KUKA KRL program: ps_b_ltb_res_c03.src, ps_b_ltb_res_c03.dat

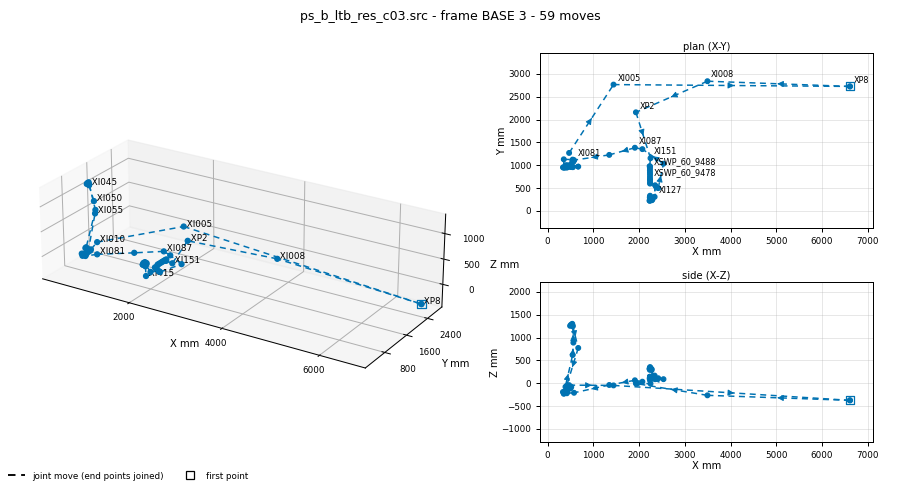
[picture p0: tool path of ps_b_ltb_res_c03.src in frame BASE 3, 59 of 59 moves have a stored position in this frame; points joined in program order, loops and branches not executed]
--- ps_b_ltb_res_c03.src ---
&ACCESS RVO1
&COMMENT Solda Atego LTB
&PARAM DISKPATH = KRC:\R1\Program\inpro_nao_mexer
DEF ps_b_ltb_res_c03( )
;FOLD INI
;FOLD SPOTTECH INI
USERSPOT(#INIT)
;ENDFOLD (SPOTTECH INI)
;FOLD GRIPPERTECH INI
USER_GRP(0,DUMMY,DUMMY,GDEFAULT)
;ENDFOLD (GRIPPERTECH INI)
  ;FOLD USER INI
    ;Make your modifications here

  ;ENDFOLD (USER INI)
;ENDFOLD (INI)

; Caracterizacao dos meios de producao
; Changes: Solda Respot - ATEGO LTB
; Versao Atual:29/10/2016
; Ferramenta: Gun C3
; Name: P13.050-R2
; optimisation

chk_w4_wechs_ok( )      ; CHECK GUN C3

;FOLD PTP P8 Vel=100 % PDAT4 Tool[4]:Gun C3 Base[3]:Atego/Axor;%{PE}%R 8.2.20,%MKUKATPBASIS,%CMOVE,%VPTP,%P 1:PTP, 2:P8, 3:, 5:100, 7:PDAT4
$BWDSTART=FALSE
PDAT_ACT=PPDAT4
FDAT_ACT=FP8
BAS(#PTP_PARAMS,100)
PTP XP8
;ENDFOLD

if MaxStandMenge (3) then
 MaxStandmengeErreicht (3)
endif

 IF (NOT(GHOST())) THEN
 if FraesAnf (3) then
 e_fraes4 ()
 endif
 ENDIF

;FOLD PTP l008 Vel=100 % P_OLP13 Tool[4]:Gun C3 Base[3]:Atego/Axor;%{PE}%R 8.2.20,%MKUKATPBASIS,%CMOVE,%VPTP,%P 1:PTP, 2:l008, 3:, 5:100, 7:P_OLP13
$BWDSTART=FALSE
PDAT_ACT=PP_OLP13
FDAT_ACT=Fl008
BAS(#PTP_PARAMS,100)
PTP Xl008
;ENDFOLD

; AGUARDA LIBERACAO PARA SOLDAR RESPOT
;FOLD OUT 3338 'R2 solda geometria Ok' State=FALSE ;%{PE}%R 8.2.20,%MKUKATPBASIS,%COUT,%VOUTX,%P 2:3338, 3:R2 solda geometria Ok, 5:FALSE, 6:
$OUT[3338]=FALSE
;ENDFOLD
;FOLD OUT 3348 'Fora area GEOBOX' State=FALSE ;%{PE}%R 8.2.20,%MKUKATPBASIS,%COUT,%VOUTX,%P 2:3348, 3:Fora area GEOBOX, 5:FALSE, 6:
$OUT[3348]=FALSE
;ENDFOLD
;FOLD OUT 3380 'Lib. p/ soldar Res Axor/Atego' State=TRUE ;%{PE}%R 8.2.20,%MKUKATPBASIS,%COUT,%VOUTX,%P 2:3380, 3:Lib. p/ soldar Res Axor/Atego, 5:TRUE, 6:
$OUT[3380]=TRUE
;ENDFOLD
;FOLD WAIT FOR ( IN 3380 'Lib. p/ soldar Res Axor/Atego' );%{PE}%R 8.2.20,%MKUKATPBASIS,%CEXT_WAIT_FOR,%VEXT_WAIT_FOR,%P 2:, 4:, 5:$IN, 6:3380, 7:Lib. p/ soldar Res Axor/Atego, 9:
WAIT FOR  ( $IN[3380] )
;ENDFOLD
;FOLD OUT 3380 'Lib. p/ soldar Res Axor/Atego' State=FALSE ;%{PE}%R 8.2.20,%MKUKATPBASIS,%COUT,%VOUTX,%P 2:3380, 3:Lib. p/ soldar Res Axor/Atego, 5:FALSE, 6:
$OUT[3380]=FALSE
;ENDFOLD

; LIGA INTERTRAVAMENTO 1 C/ R1
;FOLD Collision.Monitoring_1_On ;%{PE}%MKUKATPUSER
COLLSTOP( 1, 1 ) ;Interrupt-Controlled
;ENDFOLD

; LIGA INTERTRAVAMENTO 4 C/ R4
;FOLD Collision.Monitoring_4_On ;%{PE}%MKUKATPUSER
COLLSTOP( 4, 1 ) ;Interrupt-Controlled
;ENDFOLD

;FOLD PTP P2 CONT Vel=100 % xlarge Tool[4]:Gun C3 Base[3]:Atego/Axor;%{PE}%R 8.2.20,%MKUKATPBASIS,%CMOVE,%VPTP,%P 1:PTP, 2:P2, 3:C_DIS, 5:100, 7:xlarge
$BWDSTART=FALSE
PDAT_ACT=Pxlarge
FDAT_ACT=FP2
BAS(#PTP_PARAMS,100)
PTP XP2 C_DIS
;ENDFOLD
;FOLD PTP l151 CONT Vel=100 % large Tool[4]:Gun C3 Base[3]:Atego/Axor;%{PE}%R 8.2.20,%MKUKATPBASIS,%CMOVE,%VPTP,%P 1:PTP, 2:l151, 3:C_DIS, 5:100, 7:large
$BWDSTART=FALSE
PDAT_ACT=Plarge
FDAT_ACT=Fl151
BAS(#PTP_PARAMS,100)
PTP Xl151 C_DIS
;ENDFOLD
;FOLD PTP l146 CONT Vel=100 % fin Tool[4]:Gun C3 Base[3]:Atego/Axor;%{PE}%R 8.2.20,%MKUKATPBASIS,%CMOVE,%VPTP,%P 1:PTP, 2:l146, 3:C_DIS, 5:100, 7:fin
$BWDSTART=FALSE
PDAT_ACT=Pfin
FDAT_ACT=Fl146
BAS(#PTP_PARAMS,100)
PTP Xl146 C_DIS
;ENDFOLD

;FOLD ; SWP_60_9490;%{PE}%R 8.2.20,%MKUKATPBASIS,%CCOMMENT,%VNORMAL,%P 2:SWP_60_9490
;ENDFOLD
;FOLD PTP SWP_60_9490 vmax SPOT Gun=3 RETR CLS PgNo1=199 ACTIVE=1 Tool[4]:Gun C3 Base[3]:Atego/Axor;%{PE}%R 8.2.2,%MKUKATPSPOT,%CSPOT,%VPTP,%P 1:PTP, 2:SWP_60_9490, 3:, 5:100, 7:vmax, 10:3, 12:#FIRST, 14:#CLO, 16:199, 18:1, 20:0, 22:0, 24:1, 25:NORMAL
$BWDSTART=FALSE
PDAT_ACT=Pvmax
FDAT_ACT=FSWP_60_9490
BAS(#PTP_PARAMS,Pvmax.VEL)
S_ACT.GUN=3
S_ACT.PAIR=SDEFAULT.PAIR
S_ACT.RETR=#CLO
S_ACT.CLO_TM=1
S_ACT.PGNO1=199
S_ACT.PGNO2=SDEFAULT.PGNO2
S_ACT.PRESS1=SDEFAULT.PRESS1
S_ACT.PRESS2=SDEFAULT.PRESS2
S_READY=FALSE
PTP XSWP_60_9490
USERSPOT(#SPOT, S_ACT)
WAIT FOR S_READY
;ENDFOLD

;FOLD ; SWP_60_9488;%{PE}%R 8.2.20,%MKUKATPBASIS,%CCOMMENT,%VNORMAL,%P 2:SWP_60_9488
;ENDFOLD
;FOLD PTP SWP_60_9488 vmax SPOT Gun=3 RETR CLS PgNo1=199 ACTIVE=1 Tool[4]:Gun C3 Base[3]:Atego/Axor;%{PE}%R 8.2.2,%MKUKATPSPOT,%CSPOT,%VPTP,%P 1:PTP, 2:SWP_60_9488, 3:, 5:100, 7:vmax, 10:3, 12:#FIRST, 14:#CLO, 16:199, 18:1, 20:0, 22:0, 24:1, 25:NORMAL
$BWDSTART=FALSE
PDAT_ACT=Pvmax
FDAT_ACT=FSWP_60_9488
BAS(#PTP_PARAMS,Pvmax.VEL)
S_ACT.GUN=3
S_ACT.PAIR=SDEFAULT.PAIR
S_ACT.RETR=#CLO
S_ACT.CLO_TM=1
S_ACT.PGNO1=199
S_ACT.PGNO2=SDEFAULT.PGNO2
S_ACT.PRESS1=SDEFAULT.PRESS1
S_ACT.PRESS2=SDEFAULT.PRESS2
S_READY=FALSE
PTP XSWP_60_9488
USERSPOT(#SPOT, S_ACT)
WAIT FOR S_READY
;ENDFOLD

;FOLD ; SWP_60_9486;%{PE}%R 8.2.20,%MKUKATPBASIS,%CCOMMENT,%VNORMAL,%P 2:SWP_60_9486
;ENDFOLD
;FOLD PTP SWP_60_9486 vmax SPOT Gun=3 RETR CLS PgNo1=199 ACTIVE=1 Tool[4]:Gun C3 Base[3]:Atego/Axor;%{PE}%R 8.2.2,%MKUKATPSPOT,%CSPOT,%VPTP,%P 1:PTP, 2:SWP_60_9486, 3:, 5:100, 7:vmax, 10:3, 12:#FIRST, 14:#CLO, 16:199, 18:1, 20:0, 22:0, 24:1, 25:NORMAL
$BWDSTART=FALSE
PDAT_ACT=Pvmax
FDAT_ACT=FSWP_60_9486
BAS(#PTP_PARAMS,Pvmax.VEL)
S_ACT.GUN=3
S_ACT.PAIR=SDEFAULT.PAIR
S_ACT.RETR=#CLO
S_ACT.CLO_TM=1
S_ACT.PGNO1=199
S_ACT.PGNO2=SDEFAULT.PGNO2
S_ACT.PRESS1=SDEFAULT.PRESS1
S_ACT.PRESS2=SDEFAULT.PRESS2
S_READY=FALSE
PTP XSWP_60_9486
USERSPOT(#SPOT, S_ACT)
WAIT FOR S_READY
;ENDFOLD

;FOLD ; SWP_60_9484;%{PE}%R 8.2.20,%MKUKATPBASIS,%CCOMMENT,%VNORMAL,%P 2:SWP_60_9484
;ENDFOLD
;FOLD PTP SWP_60_9484 vmax SPOT Gun=3 RETR CLS PgNo1=199 ACTIVE=1 Tool[4]:Gun C3 Base[3]:Atego/Axor;%{PE}%R 8.2.2,%MKUKATPSPOT,%CSPOT,%VPTP,%P 1:PTP, 2:SWP_60_9484, 3:, 5:100, 7:vmax, 10:3, 12:#FIRST, 14:#CLO, 16:199, 18:1, 20:0, 22:0, 24:1, 25:NORMAL
$BWDSTART=FALSE
PDAT_ACT=Pvmax
FDAT_ACT=FSWP_60_9484
BAS(#PTP_PARAMS,Pvmax.VEL)
S_ACT.GUN=3
S_ACT.PAIR=SDEFAULT.PAIR
S_ACT.RETR=#CLO
S_ACT.CLO_TM=1
S_ACT.PGNO1=199
S_ACT.PGNO2=SDEFAULT.PGNO2
S_ACT.PRESS1=SDEFAULT.PRESS1
S_ACT.PRESS2=SDEFAULT.PRESS2
S_READY=FALSE
PTP XSWP_60_9484
USERSPOT(#SPOT, S_ACT)
WAIT FOR S_READY
;ENDFOLD

;FOLD ; SWP_60_9482;%{PE}%R 8.2.20,%MKUKATPBASIS,%CCOMMENT,%VNORMAL,%P 2:SWP_60_9482
;ENDFOLD
;FOLD PTP SWP_60_9482 vmax SPOT Gun=3 RETR CLS PgNo1=199 ACTIVE=1 Tool[4]:Gun C3 Base[3]:Atego/Axor;%{PE}%R 8.2.2,%MKUKATPSPOT,%CSPOT,%VPTP,%P 1:PTP, 2:SWP_60_9482, 3:, 5:100, 7:vmax, 10:3, 12:#FIRST, 14:#CLO, 16:199, 18:1, 20:0, 22:0, 24:1, 25:NORMAL
$BWDSTART=FALSE
PDAT_ACT=Pvmax
FDAT_ACT=FSWP_60_9482
BAS(#PTP_PARAMS,Pvmax.VEL)
S_ACT.GUN=3
S_ACT.PAIR=SDEFAULT.PAIR
S_ACT.RETR=#CLO
S_ACT.CLO_TM=1
S_ACT.PGNO1=199
S_ACT.PGNO2=SDEFAULT.PGNO2
S_ACT.PRESS1=SDEFAULT.PRESS1
S_ACT.PRESS2=SDEFAULT.PRESS2
S_READY=FALSE
PTP XSWP_60_9482
USERSPOT(#SPOT, S_ACT)
WAIT FOR S_READY
;ENDFOLD

;FOLD ; SWP_60_9480;%{PE}%R 8.2.20,%MKUKATPBASIS,%CCOMMENT,%VNORMAL,%P 2:SWP_60_9480
;ENDFOLD
;FOLD PTP SWP_60_9480 vmax SPOT Gun=3 RETR CLS PgNo1=199 ACTIVE=1 Tool[4]:Gun C3 Base[3]:Atego/Axor;%{PE}%R 8.2.2,%MKUKATPSPOT,%CSPOT,%VPTP,%P 1:PTP, 2:SWP_60_9480, 3:, 5:100, 7:vmax, 10:3, 12:#FIRST, 14:#CLO, 16:199, 18:1, 20:0, 22:0, 24:1, 25:NORMAL
$BWDSTART=FALSE
PDAT_ACT=Pvmax
FDAT_ACT=FSWP_60_9480
BAS(#PTP_PARAMS,Pvmax.VEL)
S_ACT.GUN=3
S_ACT.PAIR=SDEFAULT.PAIR
S_ACT.RETR=#CLO
S_ACT.CLO_TM=1
S_ACT.PGNO1=199
S_ACT.PGNO2=SDEFAULT.PGNO2
S_ACT.PRESS1=SDEFAULT.PRESS1
S_ACT.PRESS2=SDEFAULT.PRESS2
S_READY=FALSE
PTP XSWP_60_9480
USERSPOT(#SPOT, S_ACT)
WAIT FOR S_READY
;ENDFOLD

;FOLD ; SWP_60_9478;%{PE}%R 8.2.20,%MKUKATPBASIS,%CCOMMENT,%VNORMAL,%P 2:SWP_60_9478
;ENDFOLD
;FOLD PTP SWP_60_9478 vmax SPOT Gun=3 RETR CLS PgNo1=199 ACTIVE=1 Tool[4]:Gun C3 Base[3]:Atego/Axor;%{PE}%R 8.2.2,%MKUKATPSPOT,%CSPOT,%VPTP,%P 1:PTP, 2:SWP_60_9478, 3:, 5:100, 7:vmax, 10:3, 12:#FIRST, 14:#CLO, 16:199, 18:1, 20:0, 22:0, 24:1, 25:NORMAL
$BWDSTART=FALSE
PDAT_ACT=Pvmax
FDAT_ACT=FSWP_60_9478
BAS(#PTP_PARAMS,Pvmax.VEL)
S_ACT.GUN=3
S_ACT.PAIR=SDEFAULT.PAIR
S_ACT.RETR=#CLO
S_ACT.CLO_TM=1
S_ACT.PGNO1=199
S_ACT.PGNO2=SDEFAULT.PGNO2
S_ACT.PRESS1=SDEFAULT.PRESS1
S_ACT.PRESS2=SDEFAULT.PRESS2
S_READY=FALSE
PTP XSWP_60_9478
USERSPOT(#SPOT, S_ACT)
WAIT FOR S_READY
;ENDFOLD

;FOLD PTP l140 CONT Vel=100 % fin Tool[4]:Gun C3 Base[3]:Atego/Axor;%{PE}%R 8.2.20,%MKUKATPBASIS,%CMOVE,%VPTP,%P 1:PTP, 2:l140, 3:C_DIS, 5:100, 7:fin
$BWDSTART=FALSE
PDAT_ACT=Pfin
FDAT_ACT=Fl140
BAS(#PTP_PARAMS,100)
PTP Xl140 C_DIS
;ENDFOLD

;FOLD ; SWP_60_9474;%{PE}%R 8.2.20,%MKUKATPBASIS,%CCOMMENT,%VNORMAL,%P 2:SWP_60_9474
;ENDFOLD
;FOLD PTP SWP_60_9474 vmax SPOT Gun=3 RETR CLS PgNo1=199 ACTIVE=1 Tool[4]:Gun C3 Base[3]:Atego/Axor;%{PE}%R 8.2.2,%MKUKATPSPOT,%CSPOT,%VPTP,%P 1:PTP, 2:SWP_60_9474, 3:, 5:100, 7:vmax, 10:3, 12:#FIRST, 14:#CLO, 16:199, 18:1, 20:0, 22:0, 24:1, 25:NORMAL
$BWDSTART=FALSE
PDAT_ACT=Pvmax
FDAT_ACT=FSWP_60_9474
BAS(#PTP_PARAMS,Pvmax.VEL)
S_ACT.GUN=3
S_ACT.PAIR=SDEFAULT.PAIR
S_ACT.RETR=#CLO
S_ACT.CLO_TM=1
S_ACT.PGNO1=199
S_ACT.PGNO2=SDEFAULT.PGNO2
S_ACT.PRESS1=SDEFAULT.PRESS1
S_ACT.PRESS2=SDEFAULT.PRESS2
S_READY=FALSE
PTP XSWP_60_9474
USERSPOT(#SPOT, S_ACT)
WAIT FOR S_READY
;ENDFOLD

; LIGA INTERTRAVAMENTO 12 C/ R1
;FOLD Collision.Monitoring_AREA_6_On ;%{PE}%MKUKATPUSER
COLLSTOP( 12, 1 ) ;not Interrupt-Controlled
;ENDFOLD

;FOLD PTP l131 CONT Vel=100 % fin Tool[4]:Gun C3 Base[3]:Atego/Axor;%{PE}%R 8.2.20,%MKUKATPBASIS,%CMOVE,%VPTP,%P 1:PTP, 2:l131, 3:C_DIS, 5:100, 7:fin
$BWDSTART=FALSE
PDAT_ACT=Pfin
FDAT_ACT=Fl131
BAS(#PTP_PARAMS,100)
PTP Xl131 C_DIS
;ENDFOLD
;FOLD PTP l126 CONT Vel=100 % small Tool[4]:Gun C3 Base[3]:Atego/Axor;%{PE}%R 8.2.20,%MKUKATPBASIS,%CMOVE,%VPTP,%P 1:PTP, 2:l126, 3:C_DIS, 5:100, 7:small
$BWDSTART=FALSE
PDAT_ACT=Psmall
FDAT_ACT=Fl126
BAS(#PTP_PARAMS,100)
PTP Xl126 C_DIS
;ENDFOLD
;FOLD PTP l127 CONT Vel=100 % small Tool[4]:Gun C3 Base[3]:Atego/Axor;%{PE}%R 8.2.20,%MKUKATPBASIS,%CMOVE,%VPTP,%P 1:PTP, 2:l127, 3:C_DIS, 5:100, 7:small
$BWDSTART=FALSE
PDAT_ACT=Psmall
FDAT_ACT=Fl127
BAS(#PTP_PARAMS,100)
PTP Xl127 C_DIS
;ENDFOLD
;FOLD PTP l128 CONT Vel=100 % fin Tool[4]:Gun C3 Base[3]:Atego/Axor;%{PE}%R 8.2.20,%MKUKATPBASIS,%CMOVE,%VPTP,%P 1:PTP, 2:l128, 3:C_DIS, 5:100, 7:fin
$BWDSTART=FALSE
PDAT_ACT=Pfin
FDAT_ACT=Fl128
BAS(#PTP_PARAMS,100)
PTP Xl128 C_DIS
;ENDFOLD

;FOLD ; SWP_60_9470;%{PE}%R 8.2.20,%MKUKATPBASIS,%CCOMMENT,%VNORMAL,%P 2:SWP_60_9470
;ENDFOLD
;FOLD PTP SWP_60_9470 vmax SPOT Gun=3 RETR CLS PgNo1=199 ACTIVE=1 Tool[4]:Gun C3 Base[3]:Atego/Axor;%{PE}%R 8.2.2,%MKUKATPSPOT,%CSPOT,%VPTP,%P 1:PTP, 2:SWP_60_9470, 3:, 5:100, 7:vmax, 10:3, 12:#FIRST, 14:#CLO, 16:199, 18:1, 20:0, 22:0, 24:1, 25:NORMAL
$BWDSTART=FALSE
PDAT_ACT=Pvmax
FDAT_ACT=FSWP_60_9470
BAS(#PTP_PARAMS,Pvmax.VEL)
S_ACT.GUN=3
S_ACT.PAIR=SDEFAULT.PAIR
S_ACT.RETR=#CLO
S_ACT.CLO_TM=1
S_ACT.PGNO1=199
S_ACT.PGNO2=SDEFAULT.PGNO2
S_ACT.PRESS1=SDEFAULT.PRESS1
S_ACT.PRESS2=SDEFAULT.PRESS2
S_READY=FALSE
PTP XSWP_60_9470
USERSPOT(#SPOT, S_ACT)
WAIT FOR S_READY
;ENDFOLD

;FOLD ; SWP_60_9468;%{PE}%R 8.2.20,%MKUKATPBASIS,%CCOMMENT,%VNORMAL,%P 2:SWP_60_9468
;ENDFOLD
;FOLD PTP SWP_60_9468 vmax SPOT Gun=3 RETR CLS PgNo1=199 ACTIVE=1 Tool[4]:Gun C3 Base[3]:Atego/Axor;%{PE}%R 8.2.2,%MKUKATPSPOT,%CSPOT,%VPTP,%P 1:PTP, 2:SWP_60_9468, 3:, 5:100, 7:vmax, 10:3, 12:#FIRST, 14:#CLO, 16:199, 18:1, 20:0, 22:0, 24:1, 25:NORMAL
$BWDSTART=FALSE
PDAT_ACT=Pvmax
FDAT_ACT=FSWP_60_9468
BAS(#PTP_PARAMS,Pvmax.VEL)
S_ACT.GUN=3
S_ACT.PAIR=SDEFAULT.PAIR
S_ACT.RETR=#CLO
S_ACT.CLO_TM=1
S_ACT.PGNO1=199
S_ACT.PGNO2=SDEFAULT.PGNO2
S_ACT.PRESS1=SDEFAULT.PRESS1
S_ACT.PRESS2=SDEFAULT.PRESS2
S_READY=FALSE
PTP XSWP_60_9468
USERSPOT(#SPOT, S_ACT)
WAIT FOR S_READY
;ENDFOLD

;FOLD PTP l129 CONT Vel=100 % fin Tool[4]:Gun C3 Base[3]:Atego/Axor;%{PE}%R 8.2.20,%MKUKATPBASIS,%CMOVE,%VPTP,%P 1:PTP, 2:l129, 3:C_DIS, 5:100, 7:fin
$BWDSTART=FALSE
PDAT_ACT=Pfin
FDAT_ACT=Fl129
BAS(#PTP_PARAMS,100)
PTP Xl129 C_DIS
;ENDFOLD
;FOLD PTP l130 CONT Vel=100 % fin Tool[4]:Gun C3 Base[3]:Atego/Axor;%{PE}%R 8.2.20,%MKUKATPBASIS,%CMOVE,%VPTP,%P 1:PTP, 2:l130, 3:C_DIS, 5:100, 7:fin
$BWDSTART=FALSE
PDAT_ACT=Pfin
FDAT_ACT=Fl130
BAS(#PTP_PARAMS,100)
PTP Xl130 C_DIS
;ENDFOLD
;FOLD PTP l132 CONT Vel=100 % fin Tool[4]:Gun C3 Base[3]:Atego/Axor;%{PE}%R 8.2.20,%MKUKATPBASIS,%CMOVE,%VPTP,%P 1:PTP, 2:l132, 3:C_DIS, 5:100, 7:fin
$BWDSTART=FALSE
PDAT_ACT=Pfin
FDAT_ACT=Fl132
BAS(#PTP_PARAMS,100)
PTP Xl132 C_DIS
;ENDFOLD
;FOLD PTP l133 CONT Vel=100 % fin Tool[4]:Gun C3 Base[3]:Atego/Axor;%{PE}%R 8.2.20,%MKUKATPBASIS,%CMOVE,%VPTP,%P 1:PTP, 2:l133, 3:C_DIS, 5:100, 7:fin
$BWDSTART=FALSE
PDAT_ACT=Pfin
FDAT_ACT=Fl133
BAS(#PTP_PARAMS,100)
PTP Xl133 C_DIS
;ENDFOLD

;FOLD ; SWP_60_9466;%{PE}%R 8.2.20,%MKUKATPBASIS,%CCOMMENT,%VNORMAL,%P 2:SWP_60_9466
;ENDFOLD
;FOLD PTP SWP_60_9466 vmax SPOT Gun=3 RETR CLS PgNo1=199 ACTIVE=1 Tool[4]:Gun C3 Base[3]:Atego/Axor;%{PE}%R 8.2.2,%MKUKATPSPOT,%CSPOT,%VPTP,%P 1:PTP, 2:SWP_60_9466, 3:, 5:100, 7:vmax, 10:3, 12:#FIRST, 14:#CLO, 16:199, 18:1, 20:0, 22:0, 24:1, 25:NORMAL
$BWDSTART=FALSE
PDAT_ACT=Pvmax
FDAT_ACT=FSWP_60_9466
BAS(#PTP_PARAMS,Pvmax.VEL)
S_ACT.GUN=3
S_ACT.PAIR=SDEFAULT.PAIR
S_ACT.RETR=#CLO
S_ACT.CLO_TM=1
S_ACT.PGNO1=199
S_ACT.PGNO2=SDEFAULT.PGNO2
S_ACT.PRESS1=SDEFAULT.PRESS1
S_ACT.PRESS2=SDEFAULT.PRESS2
S_READY=FALSE
PTP XSWP_60_9466
USERSPOT(#SPOT, S_ACT)
WAIT FOR S_READY
;ENDFOLD


;FOLD PTP l134 CONT Vel=100 % fin Tool[4]:Gun C3 Base[3]:Atego/Axor;%{PE}%R 8.2.20,%MKUKATPBASIS,%CMOVE,%VPTP,%P 1:PTP, 2:l134, 3:C_DIS, 5:100, 7:fin
$BWDSTART=FALSE
PDAT_ACT=Pfin
FDAT_ACT=Fl134
BAS(#PTP_PARAMS,100)
PTP Xl134 C_DIS
;ENDFOLD
;FOLD PTP l420 CONT Vel=100 % small Tool[4]:Gun C3 Base[3]:Atego/Axor;%{PE}%R 8.2.20,%MKUKATPBASIS,%CMOVE,%VPTP,%P 1:PTP, 2:l420, 3:C_DIS, 5:100, 7:small
$BWDSTART=FALSE
PDAT_ACT=Psmall
FDAT_ACT=Fl420
BAS(#PTP_PARAMS,100)
PTP Xl420 C_DIS
;ENDFOLD
;FOLD PTP l415 CONT Vel=100 % medium Tool[4]:Gun C3 Base[3]:Atego/Axor;%{PE}%R 8.2.20,%MKUKATPBASIS,%CMOVE,%VPTP,%P 1:PTP, 2:l415, 3:C_DIS, 5:100, 7:medium
$BWDSTART=FALSE
PDAT_ACT=Pmedium
FDAT_ACT=Fl415
BAS(#PTP_PARAMS,100)
PTP Xl415 C_DIS
;ENDFOLD
;FOLD PTP l416 CONT Vel=100 % large Tool[4]:Gun C3 Base[3]:Atego/Axor;%{PE}%R 8.2.20,%MKUKATPBASIS,%CMOVE,%VPTP,%P 1:PTP, 2:l416, 3:C_DIS, 5:100, 7:large
$BWDSTART=FALSE
PDAT_ACT=Plarge
FDAT_ACT=Fl416
BAS(#PTP_PARAMS,100)
PTP Xl416 C_DIS
;ENDFOLD
;FOLD PTP l410 CONT Vel=100 % xlarge Tool[4]:Gun C3 Base[3]:Atego/Axor;%{PE}%R 8.2.20,%MKUKATPBASIS,%CMOVE,%VPTP,%P 1:PTP, 2:l410, 3:C_DIS, 5:100, 7:xlarge
$BWDSTART=FALSE
PDAT_ACT=Pxlarge
FDAT_ACT=Fl410
BAS(#PTP_PARAMS,100)
PTP Xl410 C_DIS
;ENDFOLD
;FOLD PTP l086 CONT Vel=100 % xlarge Tool[4]:Gun C3 Base[3]:Atego/Axor;%{PE}%R 8.2.20,%MKUKATPBASIS,%CMOVE,%VPTP,%P 1:PTP, 2:l086, 3:C_DIS, 5:100, 7:xlarge
$BWDSTART=FALSE
PDAT_ACT=Pxlarge
FDAT_ACT=Fl086
BAS(#PTP_PARAMS,100)
PTP Xl086 C_DIS
;ENDFOLD
;FOLD PTP l087 CONT Vel=100 % large Tool[4]:Gun C3 Base[3]:Atego/Axor;%{PE}%R 8.2.20,%MKUKATPBASIS,%CMOVE,%VPTP,%P 1:PTP, 2:l087, 3:C_DIS, 5:100, 7:large
$BWDSTART=FALSE
PDAT_ACT=Plarge
FDAT_ACT=Fl087
BAS(#PTP_PARAMS,100)
PTP Xl087 C_DIS
;ENDFOLD
;FOLD PTP l088 CONT Vel=100 % large Tool[4]:Gun C3 Base[3]:Atego/Axor;%{PE}%R 8.2.20,%MKUKATPBASIS,%CMOVE,%VPTP,%P 1:PTP, 2:l088, 3:C_DIS, 5:100, 7:large
$BWDSTART=FALSE
PDAT_ACT=Plarge
FDAT_ACT=Fl088
BAS(#PTP_PARAMS,100)
PTP Xl088 C_DIS
;ENDFOLD
;FOLD PTP l081 CONT Vel=100 % medium Tool[4]:Gun C3 Base[3]:Atego/Axor;%{PE}%R 8.2.20,%MKUKATPBASIS,%CMOVE,%VPTP,%P 1:PTP, 2:l081, 3:C_DIS, 5:100, 7:medium
$BWDSTART=FALSE
PDAT_ACT=Pmedium
FDAT_ACT=Fl081
BAS(#PTP_PARAMS,100)
PTP Xl081 C_DIS
;ENDFOLD
;FOLD PTP l076 CONT Vel=100 % fin Tool[4]:Gun C3 Base[3]:Atego/Axor;%{PE}%R 8.2.20,%MKUKATPBASIS,%CMOVE,%VPTP,%P 1:PTP, 2:l076, 3:C_DIS, 5:100, 7:fin
$BWDSTART=FALSE
PDAT_ACT=Pfin
FDAT_ACT=Fl076
BAS(#PTP_PARAMS,100)
PTP Xl076 C_DIS
;ENDFOLD

;FOLD ; SWP_60_9054;%{PE}%R 8.2.20,%MKUKATPBASIS,%CCOMMENT,%VNORMAL,%P 2:SWP_60_9054
;ENDFOLD
;FOLD PTP SWP_60_9054 vmax SPOT Gun=3 RETR CLS PgNo1=202 ACTIVE=1 Tool[4]:Gun C3 Base[3]:Atego/Axor;%{PE}%R 8.2.2,%MKUKATPSPOT,%CSPOT,%VPTP,%P 1:PTP, 2:SWP_60_9054, 3:, 5:100, 7:vmax, 10:3, 12:#FIRST, 14:#CLO, 16:202, 18:1, 20:0, 22:0, 24:1, 25:NORMAL
$BWDSTART=FALSE
PDAT_ACT=Pvmax
FDAT_ACT=FSWP_60_9054
BAS(#PTP_PARAMS,Pvmax.VEL)
S_ACT.GUN=3
S_ACT.PAIR=SDEFAULT.PAIR
S_ACT.RETR=#CLO
S_ACT.CLO_TM=1
S_ACT.PGNO1=202
S_ACT.PGNO2=SDEFAULT.PGNO2
S_ACT.PRESS1=SDEFAULT.PRESS1
S_ACT.PRESS2=SDEFAULT.PRESS2
S_READY=FALSE
PTP XSWP_60_9054
USERSPOT(#SPOT, S_ACT)
WAIT FOR S_READY
;ENDFOLD

; DESLIGA INTERTRAVAMENTO 12 C/ R1
;FOLD Collision.Monitoring_AREA_6_Off . ;%{PE}%MKUKATPUSER
COLLSTOP( 12, 2+0 )
;ENDFOLD

;FOLD ; SWP_60_9048;%{PE}%R 8.2.20,%MKUKATPBASIS,%CCOMMENT,%VNORMAL,%P 2:SWP_60_9048
;ENDFOLD
;FOLD PTP SWP_60_9048 vmax SPOT Gun=3 RETR CLS PgNo1=202 ACTIVE=1 Tool[4]:Gun C3 Base[3]:Atego/Axor;%{PE}%R 8.2.2,%MKUKATPSPOT,%CSPOT,%VPTP,%P 1:PTP, 2:SWP_60_9048, 3:, 5:100, 7:vmax, 10:3, 12:#FIRST, 14:#CLO, 16:202, 18:1, 20:0, 22:0, 24:1, 25:NORMAL
$BWDSTART=FALSE
PDAT_ACT=Pvmax
FDAT_ACT=FSWP_60_9048
BAS(#PTP_PARAMS,Pvmax.VEL)
S_ACT.GUN=3
S_ACT.PAIR=SDEFAULT.PAIR
S_ACT.RETR=#CLO
S_ACT.CLO_TM=1
S_ACT.PGNO1=202
S_ACT.PGNO2=SDEFAULT.PGNO2
S_ACT.PRESS1=SDEFAULT.PRESS1
S_ACT.PRESS2=SDEFAULT.PRESS2
S_READY=FALSE
PTP XSWP_60_9048
USERSPOT(#SPOT, S_ACT)
WAIT FOR S_READY
;ENDFOLD

;FOLD ; SWP_60_9050;%{PE}%R 8.2.20,%MKUKATPBASIS,%CCOMMENT,%VNORMAL,%P 2:SWP_60_9050
;ENDFOLD
;FOLD PTP SWP_60_9050 vmax SPOT Gun=3 RETR CLS PgNo1=202 ACTIVE=1 Tool[4]:Gun C3 Base[3]:Atego/Axor;%{PE}%R 8.2.2,%MKUKATPSPOT,%CSPOT,%VPTP,%P 1:PTP, 2:SWP_60_9050, 3:, 5:100, 7:vmax, 10:3, 12:#FIRST, 14:#CLO, 16:202, 18:1, 20:0, 22:0, 24:1, 25:NORMAL
$BWDSTART=FALSE
PDAT_ACT=Pvmax
FDAT_ACT=FSWP_60_9050
BAS(#PTP_PARAMS,Pvmax.VEL)
S_ACT.GUN=3
S_ACT.PAIR=SDEFAULT.PAIR
S_ACT.RETR=#CLO
S_ACT.CLO_TM=1
S_ACT.PGNO1=202
S_ACT.PGNO2=SDEFAULT.PGNO2
S_ACT.PRESS1=SDEFAULT.PRESS1
S_ACT.PRESS2=SDEFAULT.PRESS2
S_READY=FALSE
PTP XSWP_60_9050
USERSPOT(#SPOT, S_ACT)
WAIT FOR S_READY
;ENDFOLD

;FOLD PTP l077 CONT Vel=100 % fin Tool[4]:Gun C3 Base[3]:Atego/Axor;%{PE}%R 8.2.20,%MKUKATPBASIS,%CMOVE,%VPTP,%P 1:PTP, 2:l077, 3:C_DIS, 5:100, 7:fin
$BWDSTART=FALSE
PDAT_ACT=Pfin
FDAT_ACT=Fl077
BAS(#PTP_PARAMS,100)
PTP Xl077 C_DIS
;ENDFOLD

;FOLD ; SWP_60_9052;%{PE}%R 8.2.20,%MKUKATPBASIS,%CCOMMENT,%VNORMAL,%P 2:SWP_60_9052
;ENDFOLD
;FOLD PTP SWP_60_9052 vmax SPOT Gun=3 RETR CLS PgNo1=202 ACTIVE=1 Tool[4]:Gun C3 Base[3]:Atego/Axor;%{PE}%R 8.2.2,%MKUKATPSPOT,%CSPOT,%VPTP,%P 1:PTP, 2:SWP_60_9052, 3:, 5:100, 7:vmax, 10:3, 12:#FIRST, 14:#CLO, 16:202, 18:1, 20:0, 22:0, 24:1, 25:NORMAL
$BWDSTART=FALSE
PDAT_ACT=Pvmax
FDAT_ACT=FSWP_60_9052
BAS(#PTP_PARAMS,Pvmax.VEL)
S_ACT.GUN=3
S_ACT.PAIR=SDEFAULT.PAIR
S_ACT.RETR=#CLO
S_ACT.CLO_TM=1
S_ACT.PGNO1=202
S_ACT.PGNO2=SDEFAULT.PGNO2
S_ACT.PRESS1=SDEFAULT.PRESS1
S_ACT.PRESS2=SDEFAULT.PRESS2
S_READY=FALSE
PTP XSWP_60_9052
USERSPOT(#SPOT, S_ACT)
WAIT FOR S_READY
;ENDFOLD

; LIGA INTERTRAVAMENTO 14 C/ R5
;FOLD Collision.Monitoring_AREA_8_On ;%{PE}%MKUKATPUSER
COLLSTOP( 14, 1 ) ;not Interrupt-Controlled
;ENDFOLD

;FOLD PTP l065 CONT Vel=100 % fin Tool[4]:Gun C3 Base[3]:Atego/Axor;%{PE}%R 8.2.20,%MKUKATPBASIS,%CMOVE,%VPTP,%P 1:PTP, 2:l065, 3:C_DIS, 5:100, 7:fin
$BWDSTART=FALSE
PDAT_ACT=Pfin
FDAT_ACT=Fl065
BAS(#PTP_PARAMS,100)
PTP Xl065 C_DIS
;ENDFOLD
;FOLD PTP l060 CONT Vel=100 % small Tool[4]:Gun C3 Base[3]:Atego/Axor;%{PE}%R 8.2.20,%MKUKATPBASIS,%CMOVE,%VPTP,%P 1:PTP, 2:l060, 3:C_DIS, 5:100, 7:small
$BWDSTART=FALSE
PDAT_ACT=Psmall
FDAT_ACT=Fl060
BAS(#PTP_PARAMS,100)
PTP Xl060 C_DIS
;ENDFOLD
;FOLD PTP l055 CONT Vel=100 % xlarge Tool[4]:Gun C3 Base[3]:Atego/Axor;%{PE}%R 8.2.20,%MKUKATPBASIS,%CMOVE,%VPTP,%P 1:PTP, 2:l055, 3:C_DIS, 5:100, 7:xlarge
$BWDSTART=FALSE
PDAT_ACT=Pxlarge
FDAT_ACT=Fl055
BAS(#PTP_PARAMS,100)
PTP Xl055 C_DIS
;ENDFOLD
;FOLD PTP l050 CONT Vel=100 % xlarge Tool[4]:Gun C3 Base[3]:Atego/Axor;%{PE}%R 8.2.20,%MKUKATPBASIS,%CMOVE,%VPTP,%P 1:PTP, 2:l050, 3:C_DIS, 5:100, 7:xlarge
$BWDSTART=FALSE
PDAT_ACT=Pxlarge
FDAT_ACT=Fl050
BAS(#PTP_PARAMS,100)
PTP Xl050 C_DIS
;ENDFOLD
;FOLD PTP l045 CONT Vel=100 % fin Tool[4]:Gun C3 Base[3]:Atego/Axor;%{PE}%R 8.2.20,%MKUKATPBASIS,%CMOVE,%VPTP,%P 1:PTP, 2:l045, 3:C_DIS, 5:100, 7:fin
$BWDSTART=FALSE
PDAT_ACT=Pfin
FDAT_ACT=Fl045
BAS(#PTP_PARAMS,100)
PTP Xl045 C_DIS
;ENDFOLD

;FOLD ; SWP_60_9588;%{PE}%R 8.2.20,%MKUKATPBASIS,%CCOMMENT,%VNORMAL,%P 2:SWP_60_9588
;ENDFOLD
;FOLD PTP SWP_60_9588 vmax SPOT Gun=3 RETR CLS PgNo1=200 ACTIVE=1 Tool[4]:Gun C3 Base[3]:Atego/Axor;%{PE}%R 8.2.2,%MKUKATPSPOT,%CSPOT,%VPTP,%P 1:PTP, 2:SWP_60_9588, 3:, 5:100, 7:vmax, 10:3, 12:#FIRST, 14:#CLO, 16:200, 18:1, 20:0, 22:0, 24:1, 25:NORMAL
$BWDSTART=FALSE
PDAT_ACT=Pvmax
FDAT_ACT=FSWP_60_9588
BAS(#PTP_PARAMS,Pvmax.VEL)
S_ACT.GUN=3
S_ACT.PAIR=SDEFAULT.PAIR
S_ACT.RETR=#CLO
S_ACT.CLO_TM=1
S_ACT.PGNO1=200
S_ACT.PGNO2=SDEFAULT.PGNO2
S_ACT.PRESS1=SDEFAULT.PRESS1
S_ACT.PRESS2=SDEFAULT.PRESS2
S_READY=FALSE
PTP XSWP_60_9588
USERSPOT(#SPOT, S_ACT)
WAIT FOR S_READY
;ENDFOLD

;FOLD ; SWP_60_9586;%{PE}%R 8.2.20,%MKUKATPBASIS,%CCOMMENT,%VNORMAL,%P 2:SWP_60_9586
;ENDFOLD
;FOLD PTP SWP_60_9586 vmax SPOT Gun=3 RETR CLS PgNo1=200 ACTIVE=1 Tool[4]:Gun C3 Base[3]:Atego/Axor;%{PE}%R 8.2.2,%MKUKATPSPOT,%CSPOT,%VPTP,%P 1:PTP, 2:SWP_60_9586, 3:, 5:100, 7:vmax, 10:3, 12:#FIRST, 14:#CLO, 16:200, 18:1, 20:0, 22:0, 24:1, 25:NORMAL
$BWDSTART=FALSE
PDAT_ACT=Pvmax
FDAT_ACT=FSWP_60_9586
BAS(#PTP_PARAMS,Pvmax.VEL)
S_ACT.GUN=3
S_ACT.PAIR=SDEFAULT.PAIR
S_ACT.RETR=#CLO
S_ACT.CLO_TM=1
S_ACT.PGNO1=200
S_ACT.PGNO2=SDEFAULT.PGNO2
S_ACT.PRESS1=SDEFAULT.PRESS1
S_ACT.PRESS2=SDEFAULT.PRESS2
S_READY=FALSE
PTP XSWP_60_9586
USERSPOT(#SPOT, S_ACT)
WAIT FOR S_READY
;ENDFOLD

;FOLD ; SWP_60_9582;%{PE}%R 8.2.20,%MKUKATPBASIS,%CCOMMENT,%VNORMAL,%P 2:SWP_60_9582
;ENDFOLD
;FOLD PTP SWP_60_9582 vmax SPOT Gun=3 RETR CLS PgNo1=200 ACTIVE=1 Tool[4]:Gun C3 Base[3]:Atego/Axor;%{PE}%R 8.2.2,%MKUKATPSPOT,%CSPOT,%VPTP,%P 1:PTP, 2:SWP_60_9582, 3:, 5:100, 7:vmax, 10:3, 12:#FIRST, 14:#CLO, 16:200, 18:1, 20:0, 22:0, 24:1, 25:NORMAL
$BWDSTART=FALSE
PDAT_ACT=Pvmax
FDAT_ACT=FSWP_60_9582
BAS(#PTP_PARAMS,Pvmax.VEL)
S_ACT.GUN=3
S_ACT.PAIR=SDEFAULT.PAIR
S_ACT.RETR=#CLO
S_ACT.CLO_TM=1
S_ACT.PGNO1=200
S_ACT.PGNO2=SDEFAULT.PGNO2
S_ACT.PRESS1=SDEFAULT.PRESS1
S_ACT.PRESS2=SDEFAULT.PRESS2
S_READY=FALSE
PTP XSWP_60_9582
USERSPOT(#SPOT, S_ACT)
WAIT FOR S_READY
;ENDFOLD

;FOLD PTP l040 CONT Vel=100 % P_OLP9 Tool[4]:Gun C3 Base[3]:Atego/Axor;%{PE}%R 8.2.20,%MKUKATPBASIS,%CMOVE,%VPTP,%P 1:PTP, 2:l040, 3:C_DIS, 5:100, 7:P_OLP9
$BWDSTART=FALSE
PDAT_ACT=PP_OLP9
FDAT_ACT=Fl040
BAS(#PTP_PARAMS,100)
PTP Xl040 C_DIS
;ENDFOLD
;FOLD PTP l030 Vel=100 % P_OLP7 Tool[4]:Gun C3 Base[3]:Atego/Axor;%{PE}%R 8.2.20,%MKUKATPBASIS,%CMOVE,%VPTP,%P 1:PTP, 2:l030, 3:, 5:100, 7:P_OLP7
$BWDSTART=FALSE
PDAT_ACT=PP_OLP7
FDAT_ACT=Fl030
BAS(#PTP_PARAMS,100)
PTP Xl030
;ENDFOLD

; DESLIGA INTERTRAVAMENTO 14 C/ R5
;FOLD Collision.Monitoring_AREA_8_Off . ;%{PE}%MKUKATPUSER
COLLSTOP( 14, 2+0 )
;ENDFOLD

; LIGA INTERTRAVAMENTO 13 C/ R5
;FOLD Collision.Monitoring_AREA_7_On ;%{PE}%MKUKATPUSER
COLLSTOP( 13, 1 ) ;not Interrupt-Controlled
;ENDFOLD

;FOLD PTP l025 CONT Vel=100 % P_OLP6 Tool[4]:Gun C3 Base[3]:Atego/Axor;%{PE}%R 8.2.20,%MKUKATPBASIS,%CMOVE,%VPTP,%P 1:PTP, 2:l025, 3:C_DIS, 5:100, 7:P_OLP6
$BWDSTART=FALSE
PDAT_ACT=PP_OLP6
FDAT_ACT=Fl025
BAS(#PTP_PARAMS,100)
PTP Xl025 C_DIS
;ENDFOLD

;FOLD ; SWP_60_9076;%{PE}%R 8.2.20,%MKUKATPBASIS,%CCOMMENT,%VNORMAL,%P 2:SWP_60_9076
;ENDFOLD
;FOLD PTP SWP_60_9076 vmax SPOT Gun=3 RETR CLS PgNo1=200 ACTIVE=1 Tool[4]:Gun C3 Base[3]:Atego/Axor;%{PE}%R 8.2.2,%MKUKATPSPOT,%CSPOT,%VPTP,%P 1:PTP, 2:SWP_60_9076, 3:, 5:100, 7:vmax, 10:3, 12:#FIRST, 14:#CLO, 16:200, 18:1, 20:0, 22:0, 24:1, 25:NORMAL
$BWDSTART=FALSE
PDAT_ACT=Pvmax
FDAT_ACT=FSWP_60_9076
BAS(#PTP_PARAMS,Pvmax.VEL)
S_ACT.GUN=3
S_ACT.PAIR=SDEFAULT.PAIR
S_ACT.RETR=#CLO
S_ACT.CLO_TM=1
S_ACT.PGNO1=200
S_ACT.PGNO2=SDEFAULT.PGNO2
S_ACT.PRESS1=SDEFAULT.PRESS1
S_ACT.PRESS2=SDEFAULT.PRESS2
S_READY=FALSE
PTP XSWP_60_9076
USERSPOT(#SPOT, S_ACT)
WAIT FOR S_READY
;ENDFOLD

;FOLD ; SWP_60_9074;%{PE}%R 8.2.20,%MKUKATPBASIS,%CCOMMENT,%VNORMAL,%P 2:SWP_60_9074
;ENDFOLD
;FOLD PTP SWP_60_9074 vmax SPOT Gun=3 RETR CLS PgNo1=200 ACTIVE=1 Tool[4]:Gun C3 Base[3]:Atego/Axor;%{PE}%R 8.2.2,%MKUKATPSPOT,%CSPOT,%VPTP,%P 1:PTP, 2:SWP_60_9074, 3:, 5:100, 7:vmax, 10:3, 12:#FIRST, 14:#CLO, 16:200, 18:1, 20:0, 22:0, 24:1, 25:NORMAL
$BWDSTART=FALSE
PDAT_ACT=Pvmax
FDAT_ACT=FSWP_60_9074
BAS(#PTP_PARAMS,Pvmax.VEL)
S_ACT.GUN=3
S_ACT.PAIR=SDEFAULT.PAIR
S_ACT.RETR=#CLO
S_ACT.CLO_TM=1
S_ACT.PGNO1=200
S_ACT.PGNO2=SDEFAULT.PGNO2
S_ACT.PRESS1=SDEFAULT.PRESS1
S_ACT.PRESS2=SDEFAULT.PRESS2
S_READY=FALSE
PTP XSWP_60_9074
USERSPOT(#SPOT, S_ACT)
WAIT FOR S_READY
;ENDFOLD

;FOLD ; SWP_60_9072;%{PE}%R 8.2.20,%MKUKATPBASIS,%CCOMMENT,%VNORMAL,%P 2:SWP_60_9072
;ENDFOLD
;FOLD PTP SWP_60_9072 vmax SPOT Gun=3 RETR CLS PgNo1=200 ACTIVE=1 Tool[4]:Gun C3 Base[3]:Atego/Axor;%{PE}%R 8.2.2,%MKUKATPSPOT,%CSPOT,%VPTP,%P 1:PTP, 2:SWP_60_9072, 3:, 5:100, 7:vmax, 10:3, 12:#FIRST, 14:#CLO, 16:200, 18:1, 20:0, 22:0, 24:1, 25:NORMAL
$BWDSTART=FALSE
PDAT_ACT=Pvmax
FDAT_ACT=FSWP_60_9072
BAS(#PTP_PARAMS,Pvmax.VEL)
S_ACT.GUN=3
S_ACT.PAIR=SDEFAULT.PAIR
S_ACT.RETR=#CLO
S_ACT.CLO_TM=1
S_ACT.PGNO1=200
S_ACT.PGNO2=SDEFAULT.PGNO2
S_ACT.PRESS1=SDEFAULT.PRESS1
S_ACT.PRESS2=SDEFAULT.PRESS2
S_READY=FALSE
PTP XSWP_60_9072
USERSPOT(#SPOT, S_ACT)
WAIT FOR S_READY
;ENDFOLD

;FOLD ; SWP_60_9070;%{PE}%R 8.2.20,%MKUKATPBASIS,%CCOMMENT,%VNORMAL,%P 2:SWP_60_9070
;ENDFOLD
;FOLD PTP SWP_60_9070 vmax SPOT Gun=3 RETR OPN PgNo1=200 ACTIVE=1 Tool[4]:Gun C3 Base[3]:Atego/Axor;%{PE}%R 8.2.2,%MKUKATPSPOT,%CSPOT,%VPTP,%P 1:PTP, 2:SWP_60_9070, 3:, 5:100, 7:vmax, 10:3, 12:#FIRST, 14:#OPN, 16:200, 18:1, 20:0, 22:0, 24:1, 25:NORMAL
$BWDSTART=FALSE
PDAT_ACT=Pvmax
FDAT_ACT=FSWP_60_9070
BAS(#PTP_PARAMS,Pvmax.VEL)
S_ACT.GUN=3
S_ACT.PAIR=SDEFAULT.PAIR
S_ACT.RETR=#OPN
S_ACT.CLO_TM=1
S_ACT.PGNO1=200
S_ACT.PGNO2=SDEFAULT.PGNO2
S_ACT.PRESS1=SDEFAULT.PRESS1
S_ACT.PRESS2=SDEFAULT.PRESS2
S_READY=FALSE
PTP XSWP_60_9070
USERSPOT(#SPOT, S_ACT)
WAIT FOR S_READY
;ENDFOLD

;FOLD PTP l020 CONT Vel=100 % P_OLP5 Tool[4]:Gun C3 Base[3]:Atego/Axor;%{PE}%R 8.2.20,%MKUKATPBASIS,%CMOVE,%VPTP,%P 1:PTP, 2:l020, 3:C_DIS, 5:100, 7:P_OLP5
$BWDSTART=FALSE
PDAT_ACT=PP_OLP5
FDAT_ACT=Fl020
BAS(#PTP_PARAMS,100)
PTP Xl020 C_DIS
;ENDFOLD
;FOLD PTP l010 Vel=100 % P_OLP3 Tool[4]:Gun C3 Base[3]:Atego/Axor;%{PE}%R 8.2.20,%MKUKATPBASIS,%CMOVE,%VPTP,%P 1:PTP, 2:l010, 3:, 5:100, 7:P_OLP3
$BWDSTART=FALSE
PDAT_ACT=PP_OLP3
FDAT_ACT=Fl010
BAS(#PTP_PARAMS,100)
PTP Xl010
;ENDFOLD

; FIM DE TRABALHO RESPOT
;FOLD PULSE 3333 'R2 trabalho concluído' State=TRUE Time=3 sec;%{PE}%R 8.2.20,%MKUKATPBASIS,%COUT,%VPULSE,%P 2:3333, 3:R2 trabalho concluído, 5:TRUE, 6:, 8:3
PULSE($OUT[3333], TRUE,3)
;ENDFOLD
;FOLD OUT 3348 'Fora area GEOBOX' State=TRUE ;%{PE}%R 8.2.20,%MKUKATPBASIS,%COUT,%VOUTX,%P 2:3348, 3:Fora area GEOBOX, 5:TRUE, 6:
$OUT[3348]=TRUE
;ENDFOLD

; DESLIGA INTERTRAVAMENTO 1 C/ R1
;FOLD Collision.Monitoring_1_On ;%{PE}%MKUKATPUSER
COLLSTOP( 1, 1 ) ;Interrupt-Controlled
;ENDFOLD

; DESLIGA INTERTRAVAMENTO 4 C/ R4
;FOLD Collision.Monitoring_4_On ;%{PE}%MKUKATPUSER
COLLSTOP( 4, 1 ) ;Interrupt-Controlled
;ENDFOLD

; DESLIGA INTERTRAVAMENTO 13 C/ R5
;FOLD Collision.Monitoring_AREA_7_Off . ;%{PE}%MKUKATPUSER
COLLSTOP( 13, 2+0 )
;ENDFOLD

;FOLD PTP l005 CONT Vel=100 % xxlarge Tool[4]:Gun C3 Base[3]:Atego/Axor;%{PE}%R 8.2.20,%MKUKATPBASIS,%CMOVE,%VPTP,%P 1:PTP, 2:l005, 3:C_DIS, 5:100, 7:xxlarge
$BWDSTART=FALSE
PDAT_ACT=Pxxlarge
FDAT_ACT=Fl005
BAS(#PTP_PARAMS,100)
PTP Xl005 C_DIS
;ENDFOLD
;FOLD PTP p5 Vel=100 % vmax Tool[4]:Gun C3 Base[3]:Atego/Axor;%{PE}%R 8.2.20,%MKUKATPBASIS,%CMOVE,%VPTP,%P 1:PTP, 2:p5, 3:, 5:100, 7:vmax
$BWDSTART=FALSE
PDAT_ACT=Pvmax
FDAT_ACT=Fp5
BAS(#PTP_PARAMS,100)
PTP Xp5
;ENDFOLD

IF (NOT(GHOST())) THEN
if FraesAnf (3) then
 f_fraes4 ()
endif
ENDIF

END

--- ps_b_ltb_res_c03.dat ---
&ACCESS RVO1
&COMMENT Solda Atego LTB
&PARAM DISKPATH = KRC:\R1\Program\inpro_nao_mexer
DEFDAT ps_b_ltb_res_c03
;FOLD EXTERNAL DECLARATIONS;%{PE}%MKUKATPBASIS,%CEXT,%VCOMMON,%P
;FOLD GRIPPERTECH EXT
EXT  H50 (INT  :IN,INT  :IN,INT  :IN,GRP_TYP  :IN )
;ENDFOLD (GRIPPERTECH EXT)
;FOLD SPOTTECH EXT
EXT  USERSPOT (S_COMMAND  :IN,SPOT_TYPE  :IN )
;ENDFOLD (SPOTTECH EXT)
;FOLD BASISTECH EXT;%{PE}%MKUKATPBASIS,%CEXT,%VEXT,%P
EXT  BAS (BAS_COMMAND  :IN,REAL  :IN )
DECL INT SUCCESS
;ENDFOLD (BASISTECH EXT)
;FOLD USER EXT;%{E}%MKUKATPUSER,%CEXT,%VEXT,%P
;Make your modifications here

;ENDFOLD (USER EXT)
;ENDFOLD (EXTERNAL DECLARATIONS)
DECL FDAT Fl005={TOOL_NO 4,BASE_NO 3,IPO_FRAME #BASE,POINT2[] " "}
DECL E6POS Xl005={X 1440.43604,Y 2764.17407,Z -46.7747192,A -170.449799,B -26.6721497,C -1.85962701,S 2,T 10,E1 -4752.6748,E2 0.0,E3 0.0,E4 0.0,E5 0.0,E6 0.0}
DECL FDAT Fl010={TOOL_NO 4,BASE_NO 3,IPO_FRAME #BASE,POINT2[] " "}
DECL PDAT PP_OLP3={VEL 100.0,ACC 80.0,APO_DIST 20.0,APO_MODE #CDIS}
DECL E6POS Xl010={X 469.34079,Y 1269.60303,Z -41.1185989,A 158.067703,B 49.4165192,C 66.4640808,S 2,T 10,E1 -5700.02295,E2 0.0,E3 0.0,E4 0.0,E5 0.0,E6 0.0}
DECL FDAT Fl020={TOOL_NO 4,BASE_NO 3,IPO_FRAME #BASE,POINT2[] " "}
DECL PDAT PP_OLP5={VEL 100.0,ACC 80.0,APO_DIST 20.0,APO_MODE #CDIS}
DECL E6POS Xl020={X 515.83252,Y 999.767517,Z -78.5528564,A -147.709305,B 88.4911499,C 121.7509,S 2,T 43,E1 -5700.02295,E2 0.0,E3 0.0,E4 0.0,E5 0.0,E6 0.0}
DECL FDAT FSWP_60_9070={TOOL_NO 4,BASE_NO 3,IPO_FRAME #BASE,POINT2[] " "}
DECL E6POS XSWP_60_9070={X 502.418396,Y 998.692383,Z -106.360497,A 172.569702,B 88.708313,C 82.4837418,S 2,T 43,E1 -5700.02295,E2 0.0,E3 0.0,E4 0.0,E5 0.0,E6 0.0}
DECL FDAT FSWP_60_9072={TOOL_NO 4,BASE_NO 3,IPO_FRAME #BASE,POINT2[] " ",TQ_STATE FALSE}
DECL E6POS XSWP_60_9072={X 468.957703,Y 997.896423,Z -105.854797,A 172.576202,B 88.7087326,C 81.2132874,S 2,T 43,E1 -5700.05322,E2 0.0,E3 0.0,E4 0.0,E5 0.0,E6 0.0}
DECL FDAT FSWP_60_9074={TOOL_NO 4,BASE_NO 3,IPO_FRAME #BASE,POINT2[] " "}
DECL E6POS XSWP_60_9074={X 424.935211,Y 999.873474,Z -101.4664,A 172.584305,B 88.7084732,C 81.2202225,S 2,T 43,E1 -5700.02295,E2 0.0,E3 0.0,E4 0.0,E5 0.0,E6 0.0}
DECL FDAT FSWP_60_9076={TOOL_NO 4,BASE_NO 3,IPO_FRAME #BASE,POINT2[] " "}
DECL E6POS XSWP_60_9076={X 389.584198,Y 998.708191,Z -79.492897,A -179.567001,B 77.997467,C 89.0514069,S 2,T 43,E1 -5700.06201,E2 0.0,E3 0.0,E4 0.0,E5 0.0,E6 0.0}
DECL FDAT Fl025={TOOL_NO 4,BASE_NO 3,IPO_FRAME #BASE,POINT2[] " "}
DECL PDAT PP_OLP6={VEL 100.0,ACC 100.0,APO_DIST 20.0,APO_MODE #CDIS}
DECL E6POS Xl025={X 415.429291,Y 989.565125,Z -54.5708504,A -177.2341,B 77.9972382,C 90.649147,S 2,T 43,E1 -5700.06201,E2 0.0,E3 0.0,E4 0.0,E5 0.0,E6 0.0}
DECL FDAT Fl030={TOOL_NO 4,BASE_NO 3,IPO_FRAME #BASE,POINT2[] " "}
DECL PDAT PP_OLP7={VEL 100.0,ACC 100.0,APO_DIST 20.0,APO_MODE #CDIS}
DECL E6POS Xl030={X 668.589783,Y 970.111389,Z 772.024719,A -178.903702,B -3.26660705,C 86.3884888,S 2,T 11,E1 -5699.99609,E2 0.0,E3 0.0,E4 0.0,E5 0.0,E6 0.0}
DECL FDAT Fl040={TOOL_NO 4,BASE_NO 3,IPO_FRAME #BASE,POINT2[] " "}
DECL PDAT PP_OLP9={VEL 100.0,ACC 100.0,APO_DIST 20.0,APO_MODE #CDIS}
DECL E6POS Xl040={X 546.988098,Y 964.240479,Z 1260.33606,A -177.246307,B -55.8699989,C 86.0884018,S 2,T 11,E1 -5699.99609,E2 0.0,E3 0.0,E4 0.0,E5 0.0,E6 0.0}
DECL FDAT FSWP_60_9582={TOOL_NO 4,BASE_NO 3,IPO_FRAME #BASE,POINT2[] " "}
DECL E6POS XSWP_60_9582={X 537.534424,Y 962.133423,Z 1300.43701,A -179.627304,B -55.8536682,C 88.5657806,S 2,T 11,E1 -5699.99609,E2 0.0,E3 0.0,E4 0.0,E5 0.0,E6 0.0}
DECL FDAT FSWP_60_9586={TOOL_NO 4,BASE_NO 3,IPO_FRAME #BASE,POINT2[] " "}
DECL E6POS XSWP_60_9586={X 509.481812,Y 963.636414,Z 1279.77698,A -178.008606,B -55.8189888,C 87.2573166,S 2,T 11,E1 -5700.08008,E2 0.0,E3 0.0,E4 0.0,E5 0.0,E6 0.0}
DECL FDAT FSWP_60_9588={TOOL_NO 4,BASE_NO 3,IPO_FRAME #BASE,POINT2[] " "}
DECL E6POS XSWP_60_9588={X 490.441711,Y 966.403503,Z 1256.28503,A -174.748398,B -55.6869202,C 84.5919571,S 2,T 11,E1 -5700.00781,E2 0.0,E3 0.0,E4 0.0,E5 0.0,E6 0.0}
DECL FDAT Fl045={TOOL_NO 4,BASE_NO 3,IPO_FRAME #BASE,POINT2[] " "}
DECL E6POS Xl045={X 548.56311,Y 957.549927,Z 1245.46899,A -172.221207,B -55.5634995,C 83.9412003,S 2,T 11,E1 -5700.00781,E2 0.0,E3 0.0,E4 0.0,E5 0.0,E6 0.0}
DECL FDAT Fl050={TOOL_NO 4,BASE_NO 3,IPO_FRAME #BASE,POINT2[] " "}
DECL E6POS Xl050={X 562.548218,Y 1076.12402,Z 888.588806,A -138.753693,B -84.4868927,C 48.3102112,S 2,T 10,E1 -5699.98096,E2 0.0,E3 0.0,E4 0.0,E5 0.0,E6 0.0}
DECL FDAT Fl055={TOOL_NO 4,BASE_NO 3,IPO_FRAME #BASE,POINT2[] " "}
DECL E6POS Xl055={X 546.280518,Y 1123.396,Z 617.796997,A -56.0358505,B -85.3781662,C -35.0403786,S 2,T 10,E1 -5699.97021,E2 0.0,E3 0.0,E4 0.0,E5 0.0,E6 0.0}
DECL FDAT Fl060={TOOL_NO 4,BASE_NO 3,IPO_FRAME #BASE,POINT2[] " "}
DECL E6POS Xl060={X 352.457703,Y 1130.0,Z -221.188904,A -164.798798,B -78.1220627,C 75.1616211,S 2,T 10,E1 -5700.00391,E2 0.0,E3 0.0,E4 0.0,E5 0.0,E6 0.0}
DECL FDAT Fl065={TOOL_NO 4,BASE_NO 3,IPO_FRAME #BASE,POINT2[] " "}
DECL E6POS Xl065={X 353.910706,Y 948.556213,Z -228.998795,A -163.880905,B -78.0498581,C 74.1218185,S 2,T 11,E1 -5700.00391,E2 0.0,E3 0.0,E4 0.0,E5 0.0,E6 0.0}
DECL FDAT FSWP_60_9052={TOOL_NO 4,BASE_NO 3,IPO_FRAME #BASE,POINT2[] " ",TQ_STATE FALSE}
DECL E6POS XSWP_60_9052={X 334.658691,Y 952.987,Z -190.8508,A -170.764297,B -78.2818604,C 80.4822617,S 2,T 11,E1 -5700.00391,E2 0.0,E3 0.0,E4 0.0,E5 0.0,E6 0.0}
DECL FDAT FSWP_60_9050={TOOL_NO 4,BASE_NO 3,IPO_FRAME #BASE,POINT2[] " ",TQ_STATE FALSE}
DECL E6POS XSWP_60_9050={X 378.571106,Y 954.064392,Z -181.9561,A -175.7491,B -78.4057388,C 85.3615723,S 2,T 11,E1 -5700.00293,E2 0.0,E3 0.0,E4 0.0,E5 0.0,E6 0.0}
DECL FDAT FSWP_60_9048={TOOL_NO 4,BASE_NO 3,IPO_FRAME #BASE,POINT2[] " "}
DECL E6POS XSWP_60_9048={X 406.606598,Y 953.921875,Z -182.022598,A -175.7491,B -78.4057388,C 85.3615417,S 2,T 11,E1 -5700.01318,E2 0.0,E3 0.0,E4 0.0,E5 0.0,E6 0.0}
DECL FDAT FSWP_60_9054={TOOL_NO 4,BASE_NO 3,IPO_FRAME #BASE,POINT2[] " "}
DECL E6POS XSWP_60_9054={X 435.131805,Y 956.842224,Z -182.047699,A -175.7491,B -78.4057388,C 85.3615417,S 2,T 11,E1 -5699.99512,E2 0.0,E3 0.0,E4 0.0,E5 0.0,E6 0.0}
DECL FDAT FSWP_60_9474={TOOL_NO 4,BASE_NO 3,IPO_FRAME #BASE,POINT2[] " "}
DECL E6POS XSWP_60_9474={X 2238.87012,Y 598.833679,Z 120.386002,A -86.5505676,B -39.6951714,C -89.1793137,S 2,T 35,E1 -4500.0249,E2 0.0,E3 0.0,E4 0.0,E5 0.0,E6 0.0}
DECL FDAT Fl140={TOOL_NO 4,BASE_NO 3,IPO_FRAME #BASE,POINT2[] " "}
DECL E6POS Xl140={X 2238.51294,Y 679.724426,Z 127.631401,A -88.6769104,B -64.809639,C -90.4182205,S 2,T 35,E1 -4500.00098,E2 0.0,E3 0.0,E4 0.0,E5 0.0,E6 0.0}
DECL FDAT FSWP_60_9478={TOOL_NO 4,BASE_NO 3,IPO_FRAME #BASE,POINT2[] " "}
DECL E6POS XSWP_60_9478={X 2238.22705,Y 693.941528,Z 142.655106,A -88.063591,B -64.8049774,C -91.640007,S 2,T 35,E1 -4500.00098,E2 0.0,E3 0.0,E4 0.0,E5 0.0,E6 0.0}
DECL FDAT FSWP_60_9480={TOOL_NO 4,BASE_NO 3,IPO_FRAME #BASE,POINT2[] " "}
DECL E6POS XSWP_60_9480={X 2237.552,Y 745.543823,Z 140.875107,A -88.063591,B -64.8049774,C -91.640007,S 2,T 35,E1 -4500.04395,E2 0.0,E3 0.0,E4 0.0,E5 0.0,E6 0.0}
DECL FDAT FSWP_60_9482={TOOL_NO 4,BASE_NO 3,IPO_FRAME #BASE,POINT2[] " "}
DECL E6POS XSWP_60_9482={X 2238.17798,Y 797.964478,Z 140.041504,A -88.0616837,B -64.8083191,C -91.6423492,S 2,T 35,E1 -4500.02295,E2 0.0,E3 0.0,E4 0.0,E5 0.0,E6 0.0}
DECL FDAT FSWP_60_9484={TOOL_NO 4,BASE_NO 3,IPO_FRAME #BASE,POINT2[] " "}
DECL E6POS XSWP_60_9484={X 2237.41699,Y 842.077087,Z 139.962097,A -88.0610962,B -64.8067169,C -91.6412735,S 2,T 35,E1 -4500.00879,E2 0.0,E3 0.0,E4 0.0,E5 0.0,E6 0.0}
DECL FDAT FSWP_60_9486={TOOL_NO 4,BASE_NO 3,IPO_FRAME #BASE,POINT2[] " "}
DECL E6POS XSWP_60_9486={X 2236.19507,Y 887.221985,Z 138.260406,A -88.0627213,B -64.8068314,C -91.6403732,S 2,T 35,E1 -4500.95996,E2 0.0,E3 0.0,E4 0.0,E5 0.0,E6 0.0}
DECL FDAT FSWP_60_9488={TOOL_NO 4,BASE_NO 3,IPO_FRAME #BASE,POINT2[] " "}
DECL E6POS XSWP_60_9488={X 2237.13696,Y 932.973694,Z 139.605194,A -88.0634003,B -64.8049164,C -91.6400604,S 2,T 35,E1 -4499.99805,E2 0.0,E3 0.0,E4 0.0,E5 0.0,E6 0.0}
DECL FDAT FSWP_60_9490={TOOL_NO 4,BASE_NO 3,IPO_FRAME #BASE,POINT2[] " "}
DECL E6POS XSWP_60_9490={X 2238.30908,Y 973.484009,Z 138.175598,A -88.0585403,B -64.8054123,C -91.6460114,S 2,T 35,E1 -4499.98584,E2 0.0,E3 0.0,E4 0.0,E5 0.0,E6 0.0}
DECL BASIS_SUGG_T LAST_BASIS={POINT1[] "P0                      ",POINT2[] "P0                      ",CP_PARAMS[] "CPDAT0                  ",PTP_PARAMS[] "PDAT4                   ",CONT[] "                        ",CP_VEL[] "2.0                     ",PTP_VEL[] "100                     ",SPL_NAME[] "S0                      "}
DECL E6POS Xp5={X 6613.13379,Y 2724.13306,Z -373.284698,A 177.972397,B -19.9951,C 0.623876512,S 2,T 10,E1 199.999695,E2 0.0,E3 0.0,E4 0.0,E5 0.0,E6 0.0}
DECL FDAT Fp5={TOOL_NO 4,BASE_NO 3,IPO_FRAME #BASE,POINT2[] " ",TQ_STATE FALSE}
DECL E6POS Xl151={X 2249.06812,Y 1154.02197,Z -7.05907822,A -125.463997,B -58.1748505,C -56.5253296,S 2,T 35,E1 -4499.98584,E2 0.0,E3 0.0,E4 0.0,E5 0.0,E6 0.0}
DECL FDAT Fl151={TOOL_NO 4,BASE_NO 3,IPO_FRAME #BASE,POINT2[] " "}
DECL E6POS Xl146={X 2230.33105,Y 978.829102,Z 104.574097,A -90.7612534,B -64.7627106,C -88.9136276,S 2,T 35,E1 -4499.98584,E2 0.0,E3 0.0,E4 0.0,E5 0.0,E6 0.0}
DECL FDAT Fl146={TOOL_NO 4,BASE_NO 3,IPO_FRAME #BASE,POINT2[] " "}
DECL E6POS Xl131={X 2238.94995,Y 632.231628,Z 88.2942581,A -88.6233521,B -39.5950699,C -87.7353668,S 2,T 35,E1 -4499.99805,E2 0.0,E3 0.0,E4 0.0,E5 0.0,E6 0.0}
DECL FDAT Fl131={TOOL_NO 4,BASE_NO 3,IPO_FRAME #BASE,POINT2[] " "}
DECL E6POS Xl126={X 2350.50806,Y 562.594482,Z 88.1656036,A -85.6194992,B -39.5951004,C -87.7286072,S 2,T 35,E1 -4499.99805,E2 0.0,E3 0.0,E4 0.0,E5 0.0,E6 0.0}
DECL FDAT Fl126={TOOL_NO 4,BASE_NO 3,IPO_FRAME #BASE,POINT2[] " "}
DECL E6POS Xl086={X 2071.66797,Y 1352.54297,Z 34.8274002,A -132.405502,B -32.5161018,C -10.5114403,S 2,T 35,E1 -4700.104,E2 0.0,E3 0.0,E4 0.0,E5 0.0,E6 0.0}
DECL FDAT Fl086={TOOL_NO 4,BASE_NO 3,IPO_FRAME #BASE,POINT2[] " "}
DECL E6POS Xl081={X 576.544678,Y 1111.745,Z -208.2202,A -152.855896,B -76.8083496,C 58.5202293,S 2,T 10,E1 -5699.99512,E2 0.0,E3 0.0,E4 0.0,E5 0.0,E6 0.0}
DECL FDAT Fl081={TOOL_NO 4,BASE_NO 3,IPO_FRAME #BASE,POINT2[] " "}
DECL E6POS Xl076={X 419.960693,Y 951.812378,Z -218.835297,A -170.155197,B -78.2567673,C 79.0988235,S 2,T 11,E1 -5699.99512,E2 0.0,E3 0.0,E4 0.0,E5 0.0,E6 0.0}
DECL FDAT Fl076={TOOL_NO 4,BASE_NO 3,IPO_FRAME #BASE,POINT2[] " "}
DECL PDAT PP_OLP13={VEL 100.0,ACC 100.0,APO_DIST 0.0}
DECL E6POS Xl008={X 3494.47412,Y 2838.10693,Z -263.893005,A -178.070496,B -0.250400007,C -0.44780001,S 2,T 2,E1 -3199.99805,E2 0.0,E3 0.0,E4 0.0,E5 0.0,E6 0.0}
DECL FDAT Fl008={TOOL_NO 4,BASE_NO 3,IPO_FRAME #BASE,POINT2[] " ",TQ_STATE FALSE}
DECL E6POS XP2={X 1930.05798,Y 2158.1521,Z -5.28553009,A 177.045807,B -55.7001991,C -24.9993591,S 2,T 35,E1 -4499.23389,E2 0.0,E3 0.0,E4 0.0,E5 0.0,E6 0.0}
DECL FDAT FP2={TOOL_NO 4,BASE_NO 3,IPO_FRAME #BASE,POINT2[] " ",TQ_STATE FALSE}
DECL SPOT_SUGG_T LAST_SPOT={GUN[] "1                       ",RETR_CMD[] "#OPN                    ",CHOISE[] "#FIRST                  ",CLO_TM[] "0                       ",PGNO1[] "1                       ",PRESS1[] "0                       ",PGNO2[] "1                       ",PRESS2[] "0                       ",SPOT_PARAMS[] "NORMAL                  "}
DECL E6POS XSWP_60_9470={X 2239.24292,Y 333.695313,Z 310.066986,A 87.8133163,B -75.1693878,C 92.7297668,S 2,T 35,E1 -4499.99707,E2 0.0,E3 0.0,E4 0.0,E5 0.0,E6 0.0}
DECL FDAT FSWP_60_9470={TOOL_NO 4,BASE_NO 3,IPO_FRAME #BASE,POINT2[] " "}
DECL E6POS XSWP_60_9468={X 2239.32593,Y 282.45929,Z 349.003601,A -84.8638535,B -83.4604874,C -94.7102127,S 2,T 35,E1 -4499.99805,E2 0.0,E3 0.0,E4 0.0,E5 0.0,E6 0.0}
DECL FDAT FSWP_60_9468={TOOL_NO 4,BASE_NO 3,IPO_FRAME #BASE,POINT2[] " "}
DECL E6POS Xl420={X 2274.61694,Y 244.503296,Z 289.899414,A -118.723297,B -89.2081833,C -61.20121,S 2,T 35,E1 -4500.07324,E2 0.0,E3 0.0,E4 0.0,E5 0.0,E6 0.0}
DECL FDAT Fl420={TOOL_NO 4,BASE_NO 3,IPO_FRAME #BASE,POINT2[] " "}
DECL E6POS Xl415={X 2285.95508,Y 241.426895,Z 100.154701,A 167.887604,B -75.0239868,C 24.9231491,S 2,T 35,E1 -4500.0791,E2 0.0,E3 0.0,E4 0.0,E5 0.0,E6 0.0}
DECL FDAT Fl415={TOOL_NO 4,BASE_NO 3,IPO_FRAME #BASE,POINT2[] " "}
DECL E6POS Xl416={X 2417.54907,Y 500.388794,Z 110.236198,A -178.082901,B -63.8233604,C 21.8395309,S 2,T 35,E1 -4500.0791,E2 0.0,E3 0.0,E4 0.0,E5 0.0,E6 0.0}
DECL FDAT Fl416={TOOL_NO 4,BASE_NO 3,IPO_FRAME #BASE,POINT2[] " "}
DECL E6POS Xl410={X 2532.9021,Y 1034.12805,Z 89.4263535,A -113.278397,B -44.1855812,C -32.5207901,S 2,T 35,E1 -4500.0791,E2 0.0,E3 0.0,E4 0.0,E5 0.0,E6 0.0}
DECL FDAT Fl410={TOOL_NO 4,BASE_NO 3,IPO_FRAME #BASE,POINT2[] " "}
DECL E6POS XSWP_60_9466={X 2239.91089,Y 234.000595,Z 351.158905,A -56.0440788,B -88.7349014,C -123.509399,S 2,T 35,E1 -4500.07813,E2 0.0,E3 0.0,E4 0.0,E5 0.0,E6 0.0}
DECL FDAT FSWP_60_9466={TOOL_NO 4,BASE_NO 3,IPO_FRAME #BASE,POINT2[] " ",TQ_STATE FALSE}
DECL PDAT PPDAT4={VEL 100.0,ACC 100.0,APO_DIST 100.0}
DECL E6POS XP8={X 6609.02393,Y 2724.13794,Z -373.295807,A 177.9729,B -20.0008602,C 0.623595595,S 2,T 2,E1 450.928497,E2 0.0,E3 0.0,E4 0.0,E5 0.0,E6 0.0}
DECL FDAT FP8={TOOL_NO 4,BASE_NO 3,IPO_FRAME #BASE,POINT2[] " ",TQ_STATE FALSE}
DECL PDAT Pvmax={VEL 100.0,ACC 100.0,APO_DIST 100.0}
DECL PDAT Pfin={VEL 100.0,ACC 100.0,APO_DIST 20.0,APO_MODE #CDIS}
DECL PDAT Pxlarge={VEL 100.0,ACC 100.0,APO_DIST 500.0,APO_MODE #CDIS}
DECL PDAT Plarge={VEL 100.0,ACC 100.0,APO_DIST 200.0,APO_MODE #CDIS}
DECL PDAT Psmall={VEL 100.0,ACC 100.0,APO_DIST 50.0,APO_MODE #CDIS}
DECL E6POS Xl127={X 2339.38794,Y 309.33551,Z 167.994095,A -88.6256638,B -76.2241364,C -85.2674713,S 2,T 35,E1 -4499.99902,E2 0.0,E3 0.0,E4 0.0,E5 0.0,E6 0.0}
DECL FDAT Fl127={TOOL_NO 4,BASE_NO 3,IPO_FRAME #BASE,POINT2[] " "}
DECL E6POS Xl128={X 2234.396,Y 304.920013,Z 293.922394,A 90.8970566,B -75.1930237,C 90.5467682,S 2,T 35,E1 -4499.99805,E2 0.0,E3 0.0,E4 0.0,E5 0.0,E6 0.0}
DECL FDAT Fl128={TOOL_NO 4,BASE_NO 3,IPO_FRAME #BASE,POINT2[] " "}
DECL E6POS Xl087={X 1907.75195,Y 1383.08398,Z 65.3255386,A -128.889999,B -37.1808395,C 11.2568302,S 2,T 11,E1 -4827.78076,E2 0.0,E3 0.0,E4 0.0,E5 0.0,E6 0.0}
DECL FDAT Fl087={TOOL_NO 4,BASE_NO 3,IPO_FRAME #BASE,POINT2[] " "}
DECL E6POS Xl088={X 1347.01904,Y 1226.67505,Z -37.7420006,A -116.232399,B -49.0431709,C 21.8798695,S 2,T 11,E1 -5206.12891,E2 0.0,E3 0.0,E4 0.0,E5 0.0,E6 0.0}
DECL FDAT Fl088={TOOL_NO 4,BASE_NO 3,IPO_FRAME #BASE,POINT2[] " "}
DECL PDAT Pmedium={VEL 100.0,ACC 100.0,APO_DIST 100.0,APO_MODE #CDIS}
DECL PDAT Pxxlarge={VEL 100.0,ACC 80.0,APO_DIST 1000.0,APO_MODE #CDIS}
DECL E6POS Xl129={X 2234.80396,Y 286.454803,Z 313.757385,A -84.8638535,B -83.4604874,C -94.7102127,S 2,T 35,E1 -4499.99805,E2 0.0,E3 0.0,E4 0.0,E5 0.0,E6 0.0}
DECL FDAT Fl129={TOOL_NO 4,BASE_NO 3,IPO_FRAME #BASE,POINT2[] " "}
DECL E6POS Xl130={X 2269.59204,Y 286.731903,Z 313.432098,A -84.8638535,B -83.4604874,C -94.7102127,S 2,T 35,E1 -4499.99805,E2 0.0,E3 0.0,E4 0.0,E5 0.0,E6 0.0}
DECL FDAT Fl130={TOOL_NO 4,BASE_NO 3,IPO_FRAME #BASE,POINT2[] " "}
DECL E6POS Xl132={X 2269.33594,Y 233.462402,Z 308.926605,A -84.8637466,B -83.4604874,C -94.7103195,S 2,T 35,E1 -4499.99805,E2 0.0,E3 0.0,E4 0.0,E5 0.0,E6 0.0}
DECL FDAT Fl132={TOOL_NO 4,BASE_NO 3,IPO_FRAME #BASE,POINT2[] " "}
DECL E6POS Xl133={X 2230.47607,Y 225.487793,Z 319.069489,A 84.135643,B -85.14431,C 96.3433838,S 2,T 35,E1 -4499.99805,E2 0.0,E3 0.0,E4 0.0,E5 0.0,E6 0.0}
DECL FDAT Fl133={TOOL_NO 4,BASE_NO 3,IPO_FRAME #BASE,POINT2[] " "}
DECL E6POS Xl134={X 2230.47607,Y 225.487793,Z 319.069489,A 84.135643,B -85.14431,C 96.3433838,S 2,T 35,E1 -4499.99805,E2 0.0,E3 0.0,E4 0.0,E5 0.0,E6 0.0}
DECL FDAT Fl134={TOOL_NO 4,BASE_NO 3,IPO_FRAME #BASE,POINT2[] " "}
DECL E6POS Xl077={X 364.424591,Y 950.952087,Z -210.089996,A -171.542999,B -78.3039017,C 80.5575867,S 2,T 11,E1 -5700.00195,E2 0.0,E3 0.0,E4 0.0,E5 0.0,E6 0.0}
DECL FDAT Fl077={TOOL_NO 4,BASE_NO 3,IPO_FRAME #BASE,POINT2[] " "}
ENDDAT
